TYPE EL2521_Data :
STRUCT
	{attribute addProperty Name "Channel 1"}
	_1 :PTOChannelCompact;
END_STRUCT
END_TYPE

(* stored: Version 1.1.0.1, ProductVersion 3.1.4024.9
   DUT EL2521_Data: Id {d575ef61-7060-07a5-30c0-09a146553eed} *)
